GLOBALCONSTANTS IG2_NAME_Functions (* Industry Group 2 specific function defines *)
  (* Standard: 61499-1 *)
  (* Version 1.0, 2026-06-29, Franz Höpfinger, Demmler Andreas Fahrzeugbau *)
  PACKAGE isobus::pgn::const;
  VAR_GLOBAL CONSTANT
    F_NON_VIRTUAL_TERMINAL_DISPLAY : BYTE := 128; (* Sys: Non-specific System, Func: Non Virtual Terminal Display - An operator display connected to *)
    F_OPERATOR_CONTROLS_MACHINE_SPECIFIC : BYTE := 129; (* Sys: Non-specific System, Func: Operator Controls - Machine Specific - Operator interface *)
    F_TASK_CONTROLLER_MAPPING_COMPUTER : BYTE := 130; (* Sys: Non-specific System, Func: Task Controller (Mapping Computer) - A control function on the *)
    F_POSITION_CONTROL : BYTE := 131; (* Sys: Non-specific System, Func: Position Control - Multiple axis position control of a devices *)
    F_MACHINE_CONTROL : BYTE := 132; (* Sys: Non-specific System, Func: Machine Control - Control of outputs including adjustment of any *)
    F_FOREIGN_OBJECT_DETECTION : BYTE := 133; (* Sys: Non-specific System, Func: Foreign Object Detection - Detection of undesireable objects in *)
    F_TRACTOR_ECU : BYTE := 134; (* Sys: Non-specific System, Func: Tractor ECU - An interface unit between the tractor and the *)
    F_SEQUENCE_CONTROL_MASTER : BYTE := 135; (* Sys: Non-specific System, Func: Sequence Control Master - The master controller in the Sequence *)
    F_PRODUCT_DOSING : BYTE := 136; (* Sys: Non-specific System, Func: Product Dosing - Control function that adds an active ingredient *)
    F_PRODUCT_TREATMENT : BYTE := 137; (* Sys: Non-specific System, Func: Product Treatment - Control function that mixes a treatment to a *)
    F_RESERVED : BYTE := 138; (* Sys: Non-specific System, Func: reserved - reserved, pending discussion and approval of an "all *)
    F_DATA_LOGGER : BYTE := 139; (* Sys: Non-specific System, Func: Data Logger - Data logger as defined in ISO11783-10 for non-task *)
    F_DECISION_SUPPORT : BYTE := 140; (* Sys: Non-specific System, Func: Decision Support - A control function which is used by the *)
    F_LIGHTING_CONTROLLER : BYTE := 141; (* Sys: Non-specific System, Func: Lighting Controller - Control function that controls electrical *)
    F_TIM_SERVER : BYTE := 142; (* Sys: Non-specific System, Func: TIM Server - Control function that represents a Tractor Implement *)
    F_NOT_AVAILABLE : BYTE := 255; (* Sys: Non-specific System, Func: Not Available - This assignment can be used until an explicit *)
    F_TRACTOR_AUXILIARY_VALVE_CONTROL : BYTE := 129; (* Sys: Tractor, Func: Auxiliary Valve Control - Control of addressed tractor mounted auxiliary *)
    F_TRACTOR_REAR_HITCH_CONTROL : BYTE := 130; (* Sys: Tractor, Func: Rear Hitch Control - Control of the rear hitch of an agricultural tractor *)
    F_TRACTOR_FRONT_HITCH_CONTROL : BYTE := 131; (* Sys: Tractor, Func: Front Hitch Control - Control of the front hitch of an agricultural tractor *)
    F_TRACTOR_TRACTOR_MACHINE_CONTROL : BYTE := 132; (* Sys: Tractor, Func: Tractor Machine Control - Control of outputs including adjustment of any *)
    F_TRACTOR_CENTER_HITCH_CONTROL : BYTE := 134; (* Sys: Tractor, Func: Center Hitch Control - Control of center hitch of an agricultural tractor *)
    F_TRACTOR_NOT_AVAILABLE : BYTE := 255; (* Sys: Tractor, Func: Not Available - This assignment can be used until an explicit function has *)
    F_TILLAGE_TILLAGE_MACHINE_CONTROL : BYTE := 132; (* Sys: Tillage, Func: Tillage Machine Control - Control of outputs including adjustment of any *)
    F_TILLAGE_TILLAGE_DEPTH_CONTROL : BYTE := 135; (* Sys: Tillage, Func: Tillage Depth Control - Control of the depth of the tillage tool in the soil *)
    F_TILLAGE_FRAME_CONTROL : BYTE := 136; (* Sys: Tillage, Func: Frame Control - Control of the folding and unfolding of the frame of the *)
    F_TILLAGE_NOT_AVAILABLE : BYTE := 255; (* Sys: Tillage, Func: Not Available - This assignment can be used until an explicit function has *)
    F_SECONDARY_TILLAGE_SECONDARY_TILLAGE_MACHINE_CONTROL : BYTE := 132; (* Sys: Secondary Tillage, Func: Secondary Tillage Machine Control - Control of outputs including *)
    F_SECONDARY_TILLAGE_SECONDARY_TILLAGE_DEPTH_CONTROL : BYTE := 135; (* Sys: Secondary Tillage, Func: Secondary Tillage Depth Control - Control of the depth of the *)
    F_SECONDARY_TILLAGE_FRAME_CONTROL : BYTE := 136; (* Sys: Secondary Tillage, Func: Frame Control - Control of the folding and unfolding of the frame *)
    F_SECONDARY_TILLAGE_NOT_AVAILABLE : BYTE := 255; (* Sys: Secondary Tillage, Func: Not Available - This assignment can be used until an explicit *)
    F_PLANTERS_SEEDERS_SEED_RATE_CONTROL : BYTE := 128; (* Sys: Planters/Seeders, Func: Seed Rate Control - Control of the rate of the product placed in the *)
    F_PLANTERS_SEEDERS_SECTION_ON_OFF_CONTROL : BYTE := 129; (* Sys: Planters/Seeders, Func: Section On/Off Control - On/Off control of individual sections *)
    F_PLANTERS_SEEDERS_POSITION_CONTROL : BYTE := 131; (* Sys: Planters/Seeders, Func: Position Control - Multiple axis control of an application boom in *)
    F_PLANTERS_SEEDERS_PLANTERS_SEEDERS_MACHINE_CONTROL : BYTE := 132; (* Sys: Planters/Seeders, Func: Planters/ Seeders Machine Control - Control of outputs including *)
    F_PLANTERS_SEEDERS_PRODUCT_FLOW : BYTE := 133; (* Sys: Planters/Seeders, Func: Product Flow - Measuring function to monitor the current product *)
    F_PLANTERS_SEEDERS_PRODUCT_LEVEL : BYTE := 134; (* Sys: Planters/Seeders, Func: Product Level - Measuring function to monitor the current product *)
    F_PLANTERS_SEEDERS_DEPTH_CONTROL : BYTE := 135; (* Sys: Planters/Seeders, Func: Depth Control - Control of the depth of seed/tuber placement in the *)
    F_PLANTERS_SEEDERS_FRAME_CONTROL : BYTE := 136; (* Sys: Planters/Seeders, Func: Frame Control - Control of the folding and unfolding of the frame of *)
    F_PLANTERS_SEEDERS_DOWN_PRESSURE : BYTE := 137; (* Sys: Planters/Seeders, Func: Down Pressure - Control of the ground contact pressure on the *)
    F_PLANTERS_SEEDERS_NOT_AVAILABLE : BYTE := 255; (* Sys: Planters/Seeders, Func: Not Available - This assignment can be used until an explicit *)
    F_FERTILIZERS_FERTILIZE_RATE_CONTROL : BYTE := 128; (* Sys: Fertilizers, Func: Fertilize Rate Control - Control of the rate of product placed on or in *)
    F_FERTILIZERS_SECTION_ON_OFF_CONTROL : BYTE := 129; (* Sys: Fertilizers, Func: Section On/Off Control - On/Off control of individual sections *)
    F_FERTILIZERS_PRODUCT_PRESSURE : BYTE := 130; (* Sys: Fertilizers, Func: Product Pressure - Monitoring of the pressure of the liquid in the *)
    F_FERTILIZERS_POSITION_CONTROL : BYTE := 131; (* Sys: Fertilizers, Func: Position Control - Multiple axis control of an application boom in the x *)
    F_FERTILIZERS_FERTILIZERS_MACHINE_CONTROL : BYTE := 132; (* Sys: Fertilizers, Func: Fertilizers Machine Control - Control of outputs including adjustment of *)
    F_FERTILIZERS_PRODUCT_FLOW : BYTE := 133; (* Sys: Fertilizers, Func: Product Flow - Measuring function to monitor the current product flow. *)
    F_FERTILIZERS_PRODUCT_LEVEL : BYTE := 134; (* Sys: Fertilizers, Func: Product Level - Measuring function to monitor the current product level *)
    F_FERTILIZERS_HEIGHT_DEPTH_CONTROL : BYTE := 135; (* Sys: Fertilizers, Func: Height/Depth Control - Control of the height of the implement boom *)
    F_FERTILIZERS_FRAME_CONTROL : BYTE := 136; (* Sys: Fertilizers, Func: Frame Control - Control of the folding and unfolding of the frame of the *)
    F_FERTILIZERS_NOT_AVAILABLE : BYTE := 255; (* Sys: Fertilizers, Func: Not Available - This assignment can be used until an explicit function *)
    F_SPRAYERS_SPRAY_RATE_CONTROL : BYTE := 128; (* Sys: Sprayers, Func: Spray Rate Control - Control of the rate of crop protection product applied *)
    F_SPRAYERS_SECTION_ON_OFF_CONTROL : BYTE := 129; (* Sys: Sprayers, Func: Section On/Off Control - On/Off control of individual sections *)
    F_SPRAYERS_PRODUCT_PRESSURE : BYTE := 130; (* Sys: Sprayers, Func: Product Pressure - Monitoring of the pressure of the product in the delivery *)
    F_SPRAYERS_POSITION_CONTROL : BYTE := 131; (* Sys: Sprayers, Func: Position Control - Multiple axis control of an application boom in the x & y *)
    F_SPRAYERS_SPRAYERS_MACHINE_CONTROL : BYTE := 132; (* Sys: Sprayers, Func: Sprayers Machine Control - Control of outputs including adjustment of any *)
    F_SPRAYERS_PRODUCT_FLOW : BYTE := 133; (* Sys: Sprayers, Func: Product Flow - Measuring function to monitor the current product flow *)
    F_SPRAYERS_PRODUCT_LEVEL : BYTE := 134; (* Sys: Sprayers, Func: Product Level - Measuring function to monitor the current product level in *)
    F_SPRAYERS_BOOM_HEIGHT_CONTROL : BYTE := 135; (* Sys: Sprayers, Func: Boom Height Control - Control of the height of the boom above the surface of *)
    F_SPRAYERS_FRAME_CONTROL : BYTE := 136; (* Sys: Sprayers, Func: Frame Control - Control of the folding and unfolding of the frame of the *)
    F_SPRAYERS_NOT_AVAILABLE : BYTE := 255; (* Sys: Sprayers, Func: Not Available - This assignment can be used until an explicit function has *)
    F_HARVESTERS_TAILING_MONITOR : BYTE := 128; (* Sys: Harvesters, Func: Tailing Monitor - Measuring system to monitor the quantity of unthreshed *)
    F_HARVESTERS_HEADER_CONTROL : BYTE := 129; (* Sys: Harvesters, Func: Header Control - Control of the headers reel height and rotation and *)
    F_HARVESTERS_PRODUCT_LOSS_MONITOR : BYTE := 130; (* Sys: Harvesters, Func: Product Loss Monitor - Measuring system to monitor the amount of grain *)
    F_HARVESTERS_PRODUCT_MOISTURE : BYTE := 131; (* Sys: Harvesters, Func: Product Moisture - Measuring system to monitor the moisture content of the *)
    F_HARVESTERS_HARVESTER_MACHINE_CONTROL : BYTE := 132; (* Sys: Harvesters, Func: Harvester Machine Control - Control of outputs including adjustment of any *)
    F_HARVESTERS_PRODUCT_FLOW : BYTE := 133; (* Sys: Harvesters, Func: Product Flow - Measuring function to monitor the rate of the grain flow *)
    F_HARVESTERS_PRODUCT_LEVEL : BYTE := 134; (* Sys: Harvesters, Func: Product Level - Measuring function to monitor the grain level in the *)
    F_HARVESTERS_HEADER_HEIGHT_CONTROL : BYTE := 135; (* Sys: Harvesters, Func: Header Height Control - Control of the height of cutter bar above the *)
    F_HARVESTERS_NOT_AVAILABLE : BYTE := 255; (* Sys: Harvesters, Func: Not Available - This assignment can be used until an explicit function has *)
    F_ROOT_HARVESTERS_ROOT_HARVESTERS_MACHINE_CONTROL : BYTE := 132; (* Sys: Root Harvesters, Func: Root Harvesters Machine Control - Control of outputs including *)
    F_ROOT_HARVESTERS_PRODUCT_FLOW : BYTE := 133; (* Sys: Root Harvesters, Func: Product Flow - Measuring function to monitor the product flow into *)
    F_ROOT_HARVESTERS_PRODUCT_LEVEL : BYTE := 134; (* Sys: Root Harvesters, Func: Product Level - Measuring function to monitor the product level in *)
    F_ROOT_HARVESTERS_DEPTH_CONTROL : BYTE := 135; (* Sys: Root Harvesters, Func: Depth Control - Control of the depth of the harvestors lifter shares *)
    F_ROOT_HARVESTERS_NOT_AVAILABLE : BYTE := 255; (* Sys: Root Harvesters, Func: Not Available - This assignment can be used until an explicit *)
    F_FORAGE_TWINE_WRAPPER_CONTROL : BYTE := 128; (* Sys: Forage, Func: Twine Wrapper Control - Control of the wrapping of twine around a bale before *)
    F_FORAGE_PRODUCT_PACKAGING_CONTROL : BYTE := 129; (* Sys: Forage, Func: Product Packaging Control - Control of packaging process for the forage *)
    F_FORAGE_PRODUCT_MOISTURE : BYTE := 131; (* Sys: Forage, Func: Product Moisture - Measuring system to monitor the moisture of the forage *)
    F_FORAGE_FORAGE_MACHINE_CONTROL : BYTE := 132; (* Sys: Forage, Func: Forage Machine Control - Control of outputs including adjustment of ancillary *)
    F_FORAGE_PRODUCT_FLOW : BYTE := 133; (* Sys: Forage, Func: Product Flow - Measuring function to monitor the product flow through the *)
    F_FORAGE_WORKING_HEIGHT_CONTROL : BYTE := 135; (* Sys: Forage, Func: Working Height Control - Control of the height of cutting header above the *)
    F_FORAGE_NOT_AVAILABLE : BYTE := 255; (* Sys: Forage, Func: Not Available - This assignment can be used until an explicit function has *)
    F_IRRIGATION_NOT_AVAILABLE : BYTE := 255; (* Sys: Irrigation, Func: Not Available - This assignment can be used until an explicit function has *)
    F_TRANSPORT_TRAILER_TRANSPORT_MACHINE_CONTROL : BYTE := 132; (* Sys: Transport/Trailer, Func: Transport Machine Control - Control of outputs including adjustment *)
    F_TRANSPORT_TRAILER_UNLOAD_CONTROL : BYTE := 136; (* Sys: Transport/Trailer, Func: Unload Control - Control of trailer unloading process *)
    F_TRANSPORT_TRAILER_NOT_AVAILABLE : BYTE := 255; (* Sys: Transport/Trailer, Func: Not Available - This assignment can be used until an explicit *)
    F_FARM_YARD_OPERATIONS_NOT_AVAILABLE : BYTE := 255; (* Sys: Farm Yard Operations, Func: Not Available - This assignment can be used until an explicit *)
    F_POWERED_AUXILIARY_DEVICES_POWERED_DEVICES_MACHINE_CONTROL : BYTE := 132; (* Sys: Powered Auxiliary Devices, Func: Powered Devices Machine Control - Control of outputs *)
    F_POWERED_AUXILIARY_DEVICES_NOT_AVAILABLE : BYTE := 255; (* Sys: Powered Auxiliary Devices, Func: Not Available - This assignment can be used until an *)
    F_SPECIAL_CROPS_SPECIAL_CROP_MACHINE_CONTROL : BYTE := 132; (* Sys: Special Crops, Func: Special Crop Machine Control - Control of outputs including adjustment *)
    F_SPECIAL_CROPS_NOT_AVAILABLE : BYTE := 255; (* Sys: Special Crops, Func: Not Available - This assignment can be used until an explicit function *)
    F_EARTH_WORK_MATERIAL_RATE_CONTROL : BYTE := 128; (* Sys: Earth Work, Func: Material Rate Control - Control of the rate the material is processed. *)
    F_EARTH_WORK_EARTHWORKS_MACHINE_CONTROL : BYTE := 132; (* Sys: Earth Work, Func: Earthworks Machine Control - Control of outputs including adjustment of *)
    F_EARTH_WORK_MATERIAL_FLOW : BYTE := 133; (* Sys: Earth Work, Func: Material Flow - Measuring function to monitor the material flow *)
    F_EARTH_WORK_MATERIAL_LEVEL : BYTE := 134; (* Sys: Earth Work, Func: Material Level - Measuring function to monitor the material level *)
    F_EARTH_WORK_DEPTH_CONTROL : BYTE := 135; (* Sys: Earth Work, Func: Depth Control - Control of working depth *)
    F_EARTH_WORK_NOT_AVAILABLE : BYTE := 255; (* Sys: Earth Work, Func: Not Available - This assignment can be used until an explicit function has *)
    F_SKIDDER_SKIDDER_MACHINE_CONTROL : BYTE := 132; (* Sys: Skidder, Func: Skidder Machine Control - Control of outputs including adjustment of any *)
    F_SKIDDER_NOT_AVAILABLE : BYTE := 255; (* Sys: Skidder, Func: Not Available - This assignment can be used until an explicit function has *)
    F_SENSOR_SYSTEMS_GUIDANCE_FEELER : BYTE := 128; (* Sys: Sensor Systems, Func: Guidance Feeler - Mechanical function for determining row position in *)
    F_SENSOR_SYSTEMS_CAMERA_SYSTEM : BYTE := 129; (* Sys: Sensor Systems, Func: Camera System - Provides images or processed data for control *)
    F_SENSOR_SYSTEMS_CROP_SCOUTING : BYTE := 130; (* Sys: Sensor Systems, Func: Crop Scouting - Measures vegetation parameters in a standing crop *)
    F_SENSOR_SYSTEMS_MATERIAL_PROPERTIES_SENSING : BYTE := 131; (* Sys: Sensor Systems, Func: Material Properties Sensing - Sensing system to detect material *)
    F_SENSOR_SYSTEMS_INERTIAL_MEASUREMENT_UNIT_IMU : BYTE := 132; (* Sys: Sensor Systems, Func: Inertial Measurement Unit (IMU) - A sensor unit providing inertial *)
    F_SENSOR_SYSTEMS_PRODUCT_FLOW : BYTE := 133; (* Sys: Sensor Systems, Func: Product flow - Measuring function to monitor product flow *)
    F_SENSOR_SYSTEMS_PRODUCT_LEVEL : BYTE := 134; (* Sys: Sensor Systems, Func: Product Level - Measuring function to monitor the product level in the *)
    F_SENSOR_SYSTEMS_PRODUCT_MASS : BYTE := 135; (* Sys: Sensor Systems, Func: Product Mass - Measuring function to monitor the mass of the product *)
    F_SENSOR_SYSTEMS_VIBRATION_KNOCK : BYTE := 136; (* Sys: Sensor Systems, Func: Vibration/Knock - Measuring function to determine the vibration or *)
    F_SENSOR_SYSTEMS_WEATHER_INSTRUMENTS : BYTE := 137; (* Sys: Sensor Systems, Func: Weather Instruments - The "Weather Instruments" function code shall be *)
    F_SENSOR_SYSTEMS_SOIL_SCOUTING : BYTE := 138; (* Sys: Sensor Systems, Func: Soil Scouting - Soil Sensor to measure different soil physical *)
    F_TIMBER_HARVESTERS_TIMBER_HARVESTORS_MACHINE_CONTROL : BYTE := 132; (* Sys: Timber Harvesters, Func: Timber Harvestors Machine Control - Control of outputs including *)
    F_FORWARDERS_FORWARDERS_MACHINE_CONTROL : BYTE := 132; (* Sys: Forwarders, Func: Forwarders Machine Control - Control of outputs including adjustment of *)
    F_TIMBER_LOADERS_TIMBER_LOADERS_MACHINE_CONTROL : BYTE := 132; (* Sys: Timber Loaders, Func: Timber Loaders Machine Control - Control of outputs including *)
    F_TIMBER_PROCESSING_MACHINES_TIMBER_PROCESSING_MACHINE_CONTROL : BYTE := 132; (* Sys: Timber Processing Machines, Func: Timber Processing Machine Control - Control of outputs *)
    F_MULCHERS_MULCHER_MACHINE_CONTROL : BYTE := 132; (* Sys: Mulchers, Func: Mulcher Machine Control - Control of outputs including adjustment of any *)
    F_UTILITY_VEHICLES_UTILITY_MACHINE_CONTROL : BYTE := 132; (* Sys: Utility Vehicles, Func: Utility Machine Control - Control of outputs including adjustment of *)
    F_SLURRY_MANURE_APPLICATORS_SLURRY_MANURE_RATE_CONTROL : BYTE := 128; (* Sys: Slurry/Manure Applicators, Func: Slurry/Manure Rate Control - Control of the rate of product *)
    F_SLURRY_MANURE_APPLICATORS_SECTION_ON_OFF_CONTROL : BYTE := 129; (* Sys: Slurry/Manure Applicators, Func: Section On/Off Control - On/Off control of individual *)
    F_SLURRY_MANURE_APPLICATORS_PRODUCT_PRESSURE : BYTE := 130; (* Sys: Slurry/Manure Applicators, Func: Product Pressure - Monitoring of the pressure of the *)
    F_SLURRY_MANURE_APPLICATORS_SLURRY_MANURE_MACHINE_CONTROL : BYTE := 132; (* Sys: Slurry/Manure Applicators, Func: Slurry/Manure Machine Control - Control of outputs *)
    F_SLURRY_MANURE_APPLICATORS_PRODUCT_FLOW : BYTE := 133; (* Sys: Slurry/Manure Applicators, Func: Product Flow - Measuring function to monitor the current *)
    F_SLURRY_MANURE_APPLICATORS_PRODUCT_LEVEL : BYTE := 134; (* Sys: Slurry/Manure Applicators, Func: Product Level - Measuring function to monitor the current *)
    F_SLURRY_MANURE_APPLICATORS_BOOM_HEIGHT_CONTROL : BYTE := 135; (* Sys: Slurry/Manure Applicators, Func: Boom Height Control - Control of the height of delivery *)
    F_FEEDERS_MIXERS_FEEDER_MIXER_RATE_CONTROL : BYTE := 128; (* Sys: Feeders/Mixers, Func: Feeder/Mixer Rate Control - Control of the rate of product distributed *)
    F_FEEDERS_MIXERS_SECTION_ON_OFF_CONTROL : BYTE := 129; (* Sys: Feeders/Mixers, Func: Section On/Off Control - On/Off control of individual sections, e.g. *)
    F_FEEDERS_MIXERS_PRODUCT_PRESSURE : BYTE := 130; (* Sys: Feeders/Mixers, Func: Product Pressure - Monitoring of the pressure of the product in the *)
    F_FEEDERS_MIXERS_FEEDER_MIXER_MACHINE_CONTROL : BYTE := 132; (* Sys: Feeders/Mixers, Func: Feeder/Mixer Machine Control - Control of outputs including adjustment *)
    F_FEEDERS_MIXERS_PRODUCT_FLOW : BYTE := 133; (* Sys: Feeders/Mixers, Func: Product Flow - Measuring function to monitor the current product flow. *)
    F_FEEDERS_MIXERS_PRODUCT_LEVEL : BYTE := 134; (* Sys: Feeders/Mixers, Func: Product Level - Measuring function to monitor the current product *)
    F_FEEDERS_MIXERS_BOOM_HEIGHT_CONTROL : BYTE := 135; (* Sys: Feeders/Mixers, Func: Boom Height Control - Control of the height of delivery boom above the *)
    F_WEEDERS_WEEDER_MACHINE_CONTROL : BYTE := 132; (* Sys: Weeders - Non-chemical weed control. The device class Weeders is used by devices that *)
    F_TURF_AND_LAWN_CARE_MOWERS_TURF_AND_LAWN_CARE_MOWERS_MACHINE_CONTROL : BYTE := 132; (* Sys: Turf and Lawn Care Mowers, Func: Turf and Lawn Care Mowers Machine Control - The machine *)
    F_PRODUCT_MATERIAL_HANDLING_PRODUCT_MATERIAL_HANDLING_MACHINE_CONTROL : BYTE := 132; (* Sys: Product/Material Handling, Func: Product/Material Handling Machine Control - Control of *)
    F_PRODUCT_MATERIAL_HANDLING_PRODUCT_MATERIAL_HANDLING_PRODUCT_FLOW : BYTE := 133; (* Sys: Product/Material Handling, Func: Product/Material Handling Product Flow - Measuring function *)
    F_PRODUCT_MATERIAL_HANDLING_PRODUCT_MATERIAL_HANDLING_PRODUCT_LEVEL : BYTE := 134; (* Sys: Product/Material Handling, Func: Product/Material Handling Product Level - Meauring function *)
  END_VAR
END_GLOBALCONSTANTS
